(* Schneider Machine Expert - Basic project Schneider, file version 2.5.0.0 *)
(* ProjectInformations: Name=New project *)

HARDWARE
  Cpu 0: TM221CE24T
  EthernetConfiguration: NetworkName=M221, IpAllocationMode=FixedAddress, IpAddress=192.168.137.100, SubnetMask=255.255.255.0
  SerialLineConfiguration: Baud=Baud19200, Parity=ParityEven, DataBits=DataBits8, StopBits=StopBits1, PhysicalMedium=PhysicalMediumRs485, TransmissionMode=TransmissionModeModbusRtu, SlaveId=1, Addressing=SlaveAddressing
  MastTask: UsePeriodScanMode=false, PeriodScan=100
  FastTask: Period=255
  CpuBehavior: StartingMode=StartAsPreviousState, AutoSaveRamOnEeprom=true, WatchdogPeriod=250

SYMBOLS  (address, symbol, comment, settings)
  %MW1000   BLOCK1_START_TIME_Y  "BLOCK1 Start Time Years - 21"
  %MW1001   BLOCK1_START_TIME_M  "BLOCK1 Start Time  Months- 07"
  %MW1002   BLOCK1_START_TIME_D  "BLOCK1 Start Time Days- 19"
  %MW1003   BLOCK1_START_TIME_H  "BLOCK1 Start Time Hours - 14"
  %MW1004   BLOCK1_START_TIME_MN  "BLOCK1 Start Time Minutes - 33"
  %MW1007   BLOCK1_END_TIME_Y  "BLOCK1 End Time Years - 21"
  %MW1008   BLOCK1_END_TIME_M  "BLOCK1 End Time  Months- 07"
  %MW1009   BLOCK1_END_TIME_D  "BLOCK1 End Time Days- 19"
  %MW1010   BLOCK1_END_TIME_H  "BLOCK1 End Time Hours - 14"
  %MW1011   BLOCK1_END_TIME_MN  "BLOCK1 End Time Minutes - 33"
  %MW1012   BLOCK1_EC_SP_REAL  "BLOCK1 EC Setpoint"
  %MW1014   BLOCK1_RUNTIME_MN  "BLOCK1 Running Time for Cycle in Minutes"
  %MW1016   BLOCK1_TANK1_FLW_SP_REAL  "BLOCK1 Tank 1 Fertilizer Flow Setpoint"
  %MW1018   BLOCK1_TANK2_FLW_SP_REAL  "BLOCK1 Tank 2 Fertilizer Flow Setpoint"
  %MW1020   BLOCK1_TANK3_FLW_SP_REAL  "BLOCK1 Tank 3 Fertilizer Flow Setpoint"
  %MW1022   BLOCK1_TANK4_FLW_SP_REAL  "BLOCK1 Tank 4 Fertilizer Flow Setpoint"
  %MW1024   BLOCK1_TANK5_FLW_SP_REAL  "BLOCK1 Tank 5 Fertilizer Flow Setpoint"
  %MW1026   BLOCK1_TANK6_FLW_SP_REAL  "BLOCK1 Tank 6 Fertilizer Flow Setpoint"
  %MW1028   BLOCK1_TANK7_FLW_SP_REAL  "BLOCK1 Tank 7 Fertilizer Flow Setpoint"
  %MW1030   BLOCK1_TANK8_FLW_SP_REAL  "BLOCK1 Tank 8 Fertilizer Flow Setpoint"
  %MW1032   BLOCK1_TANK9_FLW_SP_REAL  "BLOCK1 Tank 9 Fertilizer Flow Setpoint"
  %MW1034   BLOCK1_TANK10_FLW_SP_REAL  "BLOCK1 Tank 10 Fertilizer Flow Setpoint"
  %MW1051   BLOCK2_START_TIME_Y  "BLOCK2 Start Time Years - 21"
  %MW1052   BLOCK2_START_TIME_M  "BLOCK2 Start Time  Months- 07"
  %MW1053   BLOCK2_START_TIME_D  "BLOCK2 Start Time Days- 19"
  %MW1054   BLOCK2_START_TIME_H  "BLOCK2 Start Time Hours - 14"
  %MW1055   BLOCK2_START_TIME_MN  "BLOCK2 Start Time Minutes - 33"
  %MW1058   BLOCK2_END_TIME_Y  "BLOCK2 End Time Years - 21"
  %MW1059   BLOCK2_END_TIME_M  "BLOCK2 End Time  Months- 07"
  %MW1060   BLOCK2_END_TIME_D  "BLOCK2 End Time Days- 19"
  %MW1061   BLOCK2_END_TIME_H  "BLOCK2 End Time Hours - 14"
  %MW1062   BLOCK2_END_TIME_MN  "BLOCK2 End Time Minutes - 33"
  %MW1063   BLOCK2_EC_SP_REAL  "BLOCK2 EC Setpoint"
  %MW1065   BLOCK2_RUNTIME_MN  "BLOCK2 Running Time for Cycle in Minutes"
  %MW1067   BLOCK2_TANK1_FLW_SP_REAL  "BLOCK2 Tank 1 Fertilizer Flow Setpoint"
  %MW1069   BLOCK2_TANK2_FLW_SP_REAL  "BLOCK2 Tank 2 Fertilizer Flow Setpoint"
  %MW1071   BLOCK2_TANK3_FLW_SP_REAL  "BLOCK2 Tank 3 Fertilizer Flow Setpoint"
  %MW1073   BLOCK2_TANK4_FLW_SP_REAL  "BLOCK2 Tank 4 Fertilizer Flow Setpoint"
  %MW1075   BLOCK2_TANK5_FLW_SP_REAL  "BLOCK2 Tank 5 Fertilizer Flow Setpoint"
  %MW1077   BLOCK2_TANK6_FLW_SP_REAL  "BLOCK2 Tank 6 Fertilizer Flow Setpoint"
  %MW1079   BLOCK2_TANK7_FLW_SP_REAL  "BLOCK2 Tank 7 Fertilizer Flow Setpoint"
  %MW1081   BLOCK2_TANK8_FLW_SP_REAL  "BLOCK2 Tank 8 Fertilizer Flow Setpoint"
  %MW1083   BLOCK2_TANK9_FLW_SP_REAL  "BLOCK2 Tank 9 Fertilizer Flow Setpoint"
  %MW1085   BLOCK2_TANK10_FLW_SP_REAL  "BLOCK2 Tank 10 Fertilizer Flow Setpoint"
  %MW1102   BLOCK3_START_TIME_Y  "BLOCK3 Start Time Years - 21"
  %MW1103   BLOCK3_START_TIME_M  "BLOCK3 Start Time  Months- 07"
  %MW1104   BLOCK3_START_TIME_D  "BLOCK3 Start Time Days- 19"
  %MW1105   BLOCK3_START_TIME_H  "BLOCK3 Start Time Hours - 14"
  %MW1106   BLOCK3_START_TIME_MN  "BLOCK3 Start Time Minutes - 33"
  %MW1109   BLOCK3_END_TIME_Y  "BLOCK3 End Time Years - 21"
  %MW1110   BLOCK3_END_TIME_M  "BLOCK3 End Time  Months- 07"
  %MW1111   BLOCK3_END_TIME_D  "BLOCK3 End Time Days- 19"
  %MW1112   BLOCK3_END_TIME_H  "BLOCK3 End Time Hours - 14"
  %MW1113   BLOCK3_END_TIME_MN  "BLOCK3 End Time Minutes - 33"
  %MW1114   BLOCK3_EC_SP_REAL  "BLOCK3 EC Setpoint"
  %MW1116   BLOCK3_RUNTIME_MN  "BLOCK3 Running Time for Cycle in Minutes"
  %MW1118   BLOCK3_TANK1_FLW_SP_REAL  "BLOCK3 Tank 1 Fertilizer Flow Setpoint"
  %MW1120   BLOCK3_TANK2_FLW_SP_REAL  "BLOCK3 Tank 2 Fertilizer Flow Setpoint"
  %MW1122   BLOCK3_TANK3_FLW_SP_REAL  "BLOCK3 Tank 3 Fertilizer Flow Setpoint"
  %MW1124   BLOCK3_TANK4_FLW_SP_REAL  "BLOCK3 Tank 4 Fertilizer Flow Setpoint"
  %MW1126   BLOCK3_TANK5_FLW_SP_REAL  "BLOCK3 Tank 5 Fertilizer Flow Setpoint"
  %MW1128   BLOCK3_TANK6_FLW_SP_REAL  "BLOCK3 Tank 6 Fertilizer Flow Setpoint"
  %MW1130   BLOCK3_TANK7_FLW_SP_REAL  "BLOCK3 Tank 7 Fertilizer Flow Setpoint"
  %MW1132   BLOCK3_TANK8_FLW_SP_REAL  "BLOCK3 Tank 8 Fertilizer Flow Setpoint"
  %MW1134   BLOCK3_TANK9_FLW_SP_REAL  "BLOCK3 Tank 9 Fertilizer Flow Setpoint"
  %MW1136   BLOCK3_TANK10_FLW_SP_REAL  "BLOCK3 Tank 10 Fertilizer Flow Setpoint"
  %MW1153   BLOCK4_START_TIME_Y  "BLOCK4 Start Time Years - 21"
  %MW1154   BLOCK4_START_TIME_M  "BLOCK4 Start Time  Months- 07"
  %MW1155   BLOCK4_START_TIME_D  "BLOCK4 Start Time Days- 19"
  %MW1156   BLOCK4_START_TIME_H  "BLOCK4 Start Time Hours - 14"
  %MW1157   BLOCK4_START_TIME_MN  "BLOCK4 Start Time Minutes - 33"
  %MW1160   BLOCK4_END_TIME_Y  "BLOCK4 End Time Years - 21"
  %MW1161   BLOCK4_END_TIME_M  "BLOCK4 End Time  Months- 07"
  %MW1162   BLOCK4_END_TIME_D  "BLOCK4 End Time Days- 19"
  %MW1163   BLOCK4_END_TIME_H  "BLOCK4 End Time Hours - 14"
  %MW1164   BLOCK4_END_TIME_MN  "BLOCK4 End Time Minutes - 33"
  %MW1165   BLOCK4_EC_SP_REAL  "BLOCK4 EC Setpoint"
  %MW1167   BLOCK4_RUNTIME_MN  "BLOCK4 Running Time for Cycle in Minutes"
  %MW1169   BLOCK4_TANK1_FLW_SP_REAL  "BLOCK4 Tank 1 Fertilizer Flow Setpoint"
  %MW1171   BLOCK4_TANK2_FLW_SP_REAL  "BLOCK4 Tank 2 Fertilizer Flow Setpoint"
  %MW1173   BLOCK4_TANK3_FLW_SP_REAL  "BLOCK4 Tank 3 Fertilizer Flow Setpoint"
  %MW1175   BLOCK4_TANK4_FLW_SP_REAL  "BLOCK4 Tank 4 Fertilizer Flow Setpoint"
  %MW1177   BLOCK4_TANK5_FLW_SP_REAL  "BLOCK4 Tank 5 Fertilizer Flow Setpoint"
  %MW1179   BLOCK4_TANK6_FLW_SP_REAL  "BLOCK4 Tank 6 Fertilizer Flow Setpoint"
  %MW1181   BLOCK4_TANK7_FLW_SP_REAL  "BLOCK4 Tank 7 Fertilizer Flow Setpoint"
  %MW1183   BLOCK4_TANK8_FLW_SP_REAL  "BLOCK4 Tank 8 Fertilizer Flow Setpoint"
  %MW1185   BLOCK4_TANK9_FLW_SP_REAL  "BLOCK4 Tank 9 Fertilizer Flow Setpoint"
  %MW1187   BLOCK4_TANK10_FLW_SP_REAL  "BLOCK4 Tank 10 Fertilizer Flow Setpoint"
  %MW1204   BLOCK5_START_TIME_Y  "BLOCK5 Start Time Years - 21"
  %MW1205   BLOCK5_START_TIME_M  "BLOCK5 Start Time  Months- 07"
  %MW1206   BLOCK5_START_TIME_D  "BLOCK5 Start Time Days- 19"
  %MW1207   BLOCK5_START_TIME_H  "BLOCK5 Start Time Hours - 14"
  %MW1208   BLOCK5_START_TIME_MN  "BLOCK5 Start Time Minutes - 33"
  %MW1211   BLOCK5_END_TIME_Y  "BLOCK5 End Time Years - 21"
  %MW1212   BLOCK5_END_TIME_M  "BLOCK5 End Time  Months- 07"
  %MW1213   BLOCK5_END_TIME_D  "BLOCK5 End Time Days- 19"
  %MW1214   BLOCK5_END_TIME_H  "BLOCK5 End Time Hours - 14"
  %MW1215   BLOCK5_END_TIME_MN  "BLOCK5 End Time Minutes - 33"
  %MW1216   BLOCK5_EC_SP_REAL  "BLOCK5 EC Setpoint"
  %MW1218   BLOCK5_RUNTIME_MN  "BLOCK5 Running Time for Cycle in Minutes"
  %MW1220   BLOCK5_TANK1_FLW_SP_REAL  "BLOCK5 Tank 1 Fertilizer Flow Setpoint"
  %MW1222   BLOCK5_TANK2_FLW_SP_REAL  "BLOCK5 Tank 2 Fertilizer Flow Setpoint"
  %MW1224   BLOCK5_TANK3_FLW_SP_REAL  "BLOCK5 Tank 3 Fertilizer Flow Setpoint"
  %MW1226   BLOCK5_TANK4_FLW_SP_REAL  "BLOCK5 Tank 4 Fertilizer Flow Setpoint"
  %MW1228   BLOCK5_TANK5_FLW_SP_REAL  "BLOCK5 Tank 5 Fertilizer Flow Setpoint"
  %MW1230   BLOCK5_TANK6_FLW_SP_REAL  "BLOCK5 Tank 6 Fertilizer Flow Setpoint"
  %MW1232   BLOCK5_TANK7_FLW_SP_REAL  "BLOCK5 Tank 7 Fertilizer Flow Setpoint"
  %MW1234   BLOCK5_TANK8_FLW_SP_REAL  "BLOCK5 Tank 8 Fertilizer Flow Setpoint"
  %MW1236   BLOCK5_TANK9_FLW_SP_REAL  "BLOCK5 Tank 9 Fertilizer Flow Setpoint"
  %MW1238   BLOCK5_TANK10_FLW_SP_REAL  "BLOCK5 Tank 10 Fertilizer Flow Setpoint"
  %MW1255   BLOCK6_START_TIME_Y  "BLOCK6 Start Time Years - 21"
  %MW1256   BLOCK6_START_TIME_M  "BLOCK6 Start Time  Months- 07"
  %MW1257   BLOCK6_START_TIME_D  "BLOCK6 Start Time Days- 19"
  %MW1258   BLOCK6_START_TIME_H  "BLOCK6 Start Time Hours - 14"
  %MW1259   BLOCK6_START_TIME_MN  "BLOCK6 Start Time Minutes - 33"
  %MW1262   BLOCK6_END_TIME_Y  "BLOCK6 End Time Years - 21"
  %MW1263   BLOCK6_END_TIME_M  "BLOCK6 End Time  Months- 07"
  %MW1264   BLOCK6_END_TIME_D  "BLOCK6 End Time Days- 19"
  %MW1265   BLOCK6_END_TIME_H  "BLOCK6 End Time Hours - 14"
  %MW1266   BLOCK6_END_TIME_MN  "BLOCK6 End Time Minutes - 33"
  %MW1267   BLOCK6_EC_SP_REAL  "BLOCK6 EC Setpoint"
  %MW1269   BLOCK6_RUNTIME_MN  "BLOCK6 Running Time for Cycle in Minutes"
  %MW1271   BLOCK6_TANK1_FLW_SP_REAL  "BLOCK6 Tank 1 Fertilizer Flow Setpoint"
  %MW1273   BLOCK6_TANK2_FLW_SP_REAL  "BLOCK6 Tank 2 Fertilizer Flow Setpoint"
  %MW1275   BLOCK6_TANK3_FLW_SP_REAL  "BLOCK6 Tank 3 Fertilizer Flow Setpoint"
  %MW1277   BLOCK6_TANK4_FLW_SP_REAL  "BLOCK6 Tank 4 Fertilizer Flow Setpoint"
  %MW1279   BLOCK6_TANK5_FLW_SP_REAL  "BLOCK6 Tank 5 Fertilizer Flow Setpoint"
  %MW1281   BLOCK6_TANK6_FLW_SP_REAL  "BLOCK6 Tank 6 Fertilizer Flow Setpoint"
  %MW1283   BLOCK6_TANK7_FLW_SP_REAL  "BLOCK6 Tank 7 Fertilizer Flow Setpoint"
  %MW1285   BLOCK6_TANK8_FLW_SP_REAL  "BLOCK6 Tank 8 Fertilizer Flow Setpoint"
  %MW1287   BLOCK6_TANK9_FLW_SP_REAL  "BLOCK6 Tank 9 Fertilizer Flow Setpoint"
  %MW1289   BLOCK6_TANK10_FLW_SP_REAL  "BLOCK6 Tank 10 Fertilizer Flow Setpoint"
  %MW1306   BLOCK7_START_TIME_Y  "BLOCK7 Start Time Years - 21"
  %MW1307   BLOCK7_START_TIME_M  "BLOCK7 Start Time  Months- 07"
  %MW1308   BLOCK7_START_TIME_D  "BLOCK7 Start Time Days- 19"
  %MW1309   BLOCK7_START_TIME_H  "BLOCK7 Start Time Hours - 14"
  %MW1310   BLOCK7_START_TIME_MN  "BLOCK7 Start Time Minutes - 33"
  %MW1313   BLOCK7_END_TIME_Y  "BLOCK7 End Time Years - 21"
  %MW1314   BLOCK7_END_TIME_M  "BLOCK7 End Time  Months- 07"
  %MW1315   BLOCK7_END_TIME_D  "BLOCK7 End Time Days- 19"
  %MW1316   BLOCK7_END_TIME_H  "BLOCK7 End Time Hours - 14"
  %MW1317   BLOCK7_END_TIME_MN  "BLOCK7 End Time Minutes - 33"
  %MW1318   BLOCK7_EC_SP_REAL  "BLOCK7 EC Setpoint"
  %MW1320   BLOCK7_RUNTIME_MN  "BLOCK7 Running Time for Cycle in Minutes"
  %MW1322   BLOCK7_TANK1_FLW_SP_REAL  "BLOCK7 Tank 1 Fertilizer Flow Setpoint"
  %MW1324   BLOCK7_TANK2_FLW_SP_REAL  "BLOCK7 Tank 2 Fertilizer Flow Setpoint"
  %MW1326   BLOCK7_TANK3_FLW_SP_REAL  "BLOCK7 Tank 3 Fertilizer Flow Setpoint"
  %MW1328   BLOCK7_TANK4_FLW_SP_REAL  "BLOCK7 Tank 4 Fertilizer Flow Setpoint"
  %MW1330   BLOCK7_TANK5_FLW_SP_REAL  "BLOCK7 Tank 5 Fertilizer Flow Setpoint"
  %MW1332   BLOCK7_TANK6_FLW_SP_REAL  "BLOCK7 Tank 6 Fertilizer Flow Setpoint"
  %MW1334   BLOCK7_TANK7_FLW_SP_REAL  "BLOCK7 Tank 7 Fertilizer Flow Setpoint"
  %MW1336   BLOCK7_TANK8_FLW_SP_REAL  "BLOCK7 Tank 8 Fertilizer Flow Setpoint"
  %MW1338   BLOCK7_TANK9_FLW_SP_REAL  "BLOCK7 Tank 9 Fertilizer Flow Setpoint"
  %MW1340   BLOCK7_TANK10_FLW_SP_REAL  "BLOCK7 Tank 10 Fertilizer Flow Setpoint"
  %MW1357   BLOCK8_START_TIME_Y  "BLOCK8 Start Time Years - 21"
  %MW1358   BLOCK8_START_TIME_M  "BLOCK8 Start Time  Months- 07"
  %MW1359   BLOCK8_START_TIME_D  "BLOCK8 Start Time Days- 19"
  %MW1360   BLOCK8_START_TIME_H  "BLOCK8 Start Time Hours - 14"
  %MW1361   BLOCK8_START_TIME_MN  "BLOCK8 Start Time Minutes - 33"
  %MW1364   BLOCK8_END_TIME_Y  "BLOCK8 End Time Years - 21"
  %MW1365   BLOCK8_END_TIME_M  "BLOCK8 End Time  Months- 07"
  %MW1366   BLOCK8_END_TIME_D  "BLOCK8 End Time Days- 19"
  %MW1367   BLOCK8_END_TIME_H  "BLOCK8 End Time Hours - 14"
  %MW1368   BLOCK8_END_TIME_MN  "BLOCK8 End Time Minutes - 33"
  %MW1369   BLOCK8_EC_SP_REAL  "BLOCK8 EC Setpoint"
  %MW1371   BLOCK8_RUNTIME_MN  "BLOCK8 Running Time for Cycle in Minutes"
  %MW1373   BLOCK8_TANK1_FLW_SP_REAL  "BLOCK8 Tank 1 Fertilizer Flow Setpoint"
  %MW1375   BLOCK8_TANK2_FLW_SP_REAL  "BLOCK8 Tank 2 Fertilizer Flow Setpoint"
  %MW1377   BLOCK8_TANK3_FLW_SP_REAL  "BLOCK8 Tank 3 Fertilizer Flow Setpoint"
  %MW1379   BLOCK8_TANK4_FLW_SP_REAL  "BLOCK8 Tank 4 Fertilizer Flow Setpoint"
  %MW1381   BLOCK8_TANK5_FLW_SP_REAL  "BLOCK8 Tank 5 Fertilizer Flow Setpoint"
  %MW1383   BLOCK8_TANK6_FLW_SP_REAL  "BLOCK8 Tank 6 Fertilizer Flow Setpoint"
  %MW1385   BLOCK8_TANK7_FLW_SP_REAL  "BLOCK8 Tank 7 Fertilizer Flow Setpoint"
  %MW1387   BLOCK8_TANK8_FLW_SP_REAL  "BLOCK8 Tank 8 Fertilizer Flow Setpoint"
  %MW1389   BLOCK8_TANK9_FLW_SP_REAL  "BLOCK8 Tank 9 Fertilizer Flow Setpoint"
  %MW1391   BLOCK8_TANK10_FLW_SP_REAL  "BLOCK8 Tank 10 Fertilizer Flow Setpoint"
  %MW1408   BLOCK9_START_TIME_Y  "BLOCK9 Start Time Years - 21"
  %MW1409   BLOCK9_START_TIME_M  "BLOCK9 Start Time  Months- 07"
  %MW1410   BLOCK9_START_TIME_D  "BLOCK9 Start Time Days- 19"
  %MW1411   BLOCK9_START_TIME_H  "BLOCK9 Start Time Hours - 14"
  %MW1412   BLOCK9_START_TIME_MN  "BLOCK9 Start Time Minutes - 33"
  %MW1415   BLOCK9_END_TIME_Y  "BLOCK9 End Time Years - 21"
  %MW1416   BLOCK9_END_TIME_M  "BLOCK9 End Time  Months- 07"
  %MW1417   BLOCK9_END_TIME_D  "BLOCK9 End Time Days- 19"
  %MW1418   BLOCK9_END_TIME_H  "BLOCK9 End Time Hours - 14"
  %MW1419   BLOCK9_END_TIME_MN  "BLOCK9 End Time Minutes - 33"
  %MW1420   BLOCK9_EC_SP_REAL  "BLOCK9 EC Setpoint"
  %MW1422   BLOCK9_RUNTIME_MN  "BLOCK9 Running Time for Cycle in Minutes"
  %MW1424   BLOCK9_TANK1_FLW_SP_REAL  "BLOCK9 Tank 1 Fertilizer Flow Setpoint"
  %MW1426   BLOCK9_TANK2_FLW_SP_REAL  "BLOCK9 Tank 2 Fertilizer Flow Setpoint"
  %MW1428   BLOCK9_TANK3_FLW_SP_REAL  "BLOCK9 Tank 3 Fertilizer Flow Setpoint"
  %MW1430   BLOCK9_TANK4_FLW_SP_REAL  "BLOCK9 Tank 4 Fertilizer Flow Setpoint"
  %MW1432   BLOCK9_TANK5_FLW_SP_REAL  "BLOCK9 Tank 5 Fertilizer Flow Setpoint"
  %MW1434   BLOCK9_TANK6_FLW_SP_REAL  "BLOCK9 Tank 6 Fertilizer Flow Setpoint"
  %MW1436   BLOCK9_TANK7_FLW_SP_REAL  "BLOCK9 Tank 7 Fertilizer Flow Setpoint"
  %MW1438   BLOCK9_TANK8_FLW_SP_REAL  "BLOCK9 Tank 8 Fertilizer Flow Setpoint"
  %MW1440   BLOCK9_TANK9_FLW_SP_REAL  "BLOCK9 Tank 9 Fertilizer Flow Setpoint"
  %MW1442   BLOCK9_TANK10_FLW_SP_REAL  "BLOCK9 Tank 10 Fertilizer Flow Setpoint"
  %MW1459   BLOCK10_START_TIME_Y  "BLOCK10 Start Time Years - 21"
  %MW1460   BLOCK10_START_TIME_M  "BLOCK10 Start Time  Months- 07"
  %MW1461   BLOCK10_START_TIME_D  "BLOCK10 Start Time Days- 19"
  %MW1462   BLOCK10_START_TIME_H  "BLOCK10 Start Time Hours - 14"
  %MW1463   BLOCK10_START_TIME_MN  "BLOCK10 Start Time Minutes - 33"
  %MW1466   BLOCK10_END_TIME_Y  "BLOCK10 End Time Years - 21"
  %MW1467   BLOCK10_END_TIME_M  "BLOCK10 End Time  Months- 07"
  %MW1468   BLOCK10_END_TIME_D  "BLOCK10 End Time Days- 19"
  %MW1469   BLOCK10_END_TIME_H  "BLOCK10 End Time Hours - 14"
  %MW1470   BLOCK10_END_TIME_MN  "BLOCK10 End Time Minutes - 33"
  %MW1471   BLOCK10_EC_SP_REAL  "BLOCK10 EC Setpoint"
  %MW1473   BLOCK10_RUNTIME_MN  "BLOCK10 Running Time for Cycle in Minutes"
  %MW1475   BLOCK10_TANK1_FLW_SP_REAL  "BLOCK10 Tank 1 Fertilizer Flow Setpoint"
  %MW1477   BLOCK10_TANK2_FLW_SP_REAL  "BLOCK10 Tank 2 Fertilizer Flow Setpoint"
  %MW1479   BLOCK10_TANK3_FLW_SP_REAL  "BLOCK10 Tank 3 Fertilizer Flow Setpoint"
  %MW1481   BLOCK10_TANK4_FLW_SP_REAL  "BLOCK10 Tank 4 Fertilizer Flow Setpoint"
  %MW1483   BLOCK10_TANK5_FLW_SP_REAL  "BLOCK10 Tank 5 Fertilizer Flow Setpoint"
  %MW1485   BLOCK10_TANK6_FLW_SP_REAL  "BLOCK10 Tank 6 Fertilizer Flow Setpoint"
  %MW1487   BLOCK10_TANK7_FLW_SP_REAL  "BLOCK10 Tank 7 Fertilizer Flow Setpoint"
  %MW1489   BLOCK10_TANK8_FLW_SP_REAL  "BLOCK10 Tank 8 Fertilizer Flow Setpoint"
  %MW1491   BLOCK10_TANK9_FLW_SP_REAL  "BLOCK10 Tank 9 Fertilizer Flow Setpoint"
  %MW1493   BLOCK10_TANK10_FLW_SP_REAL  "BLOCK10 Tank 10 Fertilizer Flow Setpoint"
  %MW1510   BLOCK11_START_TIME_Y  "BLOCK11 Start Time Years - 21"
  %MW1511   BLOCK11_START_TIME_M  "BLOCK11 Start Time  Months- 07"
  %MW1512   BLOCK11_START_TIME_D  "BLOCK11 Start Time Days- 19"
  %MW1513   BLOCK11_START_TIME_H  "BLOCK11 Start Time Hours - 14"
  %MW1514   BLOCK11_START_TIME_MN  "BLOCK11 Start Time Minutes - 33"
  %MW1517   BLOCK11_END_TIME_Y  "BLOCK11 End Time Years - 21"
  %MW1518   BLOCK11_END_TIME_M  "BLOCK11 End Time  Months- 07"
  %MW1519   BLOCK11_END_TIME_D  "BLOCK11 End Time Days- 19"
  %MW1520   BLOCK11_END_TIME_H  "BLOCK11 End Time Hours - 14"
  %MW1521   BLOCK11_END_TIME_MN  "BLOCK11 End Time Minutes - 33"
  %MW1522   BLOCK11_EC_SP_REAL  "BLOCK11 EC Setpoint"
  %MW1524   BLOCK11_RUNTIME_MN  "BLOCK11 Running Time for Cycle in Minutes"
  %MW1526   BLOCK11_TANK1_FLW_SP_REAL  "BLOCK11 Tank 1 Fertilizer Flow Setpoint"
  %MW1528   BLOCK11_TANK2_FLW_SP_REAL  "BLOCK11 Tank 2 Fertilizer Flow Setpoint"
  %MW1530   BLOCK11_TANK3_FLW_SP_REAL  "BLOCK11 Tank 3 Fertilizer Flow Setpoint"
  %MW1532   BLOCK11_TANK4_FLW_SP_REAL  "BLOCK11 Tank 4 Fertilizer Flow Setpoint"
  %MW1534   BLOCK11_TANK5_FLW_SP_REAL  "BLOCK11 Tank 5 Fertilizer Flow Setpoint"
  %MW1536   BLOCK11_TANK6_FLW_SP_REAL  "BLOCK11 Tank 6 Fertilizer Flow Setpoint"
  %MW1538   BLOCK11_TANK7_FLW_SP_REAL  "BLOCK11 Tank 7 Fertilizer Flow Setpoint"
  %MW1540   BLOCK11_TANK8_FLW_SP_REAL  "BLOCK11 Tank 8 Fertilizer Flow Setpoint"
  %MW1542   BLOCK11_TANK9_FLW_SP_REAL  "BLOCK11 Tank 9 Fertilizer Flow Setpoint"
  %MW1544   BLOCK11_TANK10_FLW_SP_REAL  "BLOCK11 Tank 10 Fertilizer Flow Setpoint"
  %MW1561   BLOCK12_START_TIME_Y  "BLOCK12 Start Time Years - 21"
  %MW1562   BLOCK12_START_TIME_M  "BLOCK12 Start Time  Months- 07"
  %MW1563   BLOCK12_START_TIME_D  "BLOCK12 Start Time Days- 19"
  %MW1564   BLOCK12_START_TIME_H  "BLOCK12 Start Time Hours - 14"
  %MW1565   BLOCK12_START_TIME_MN  "BLOCK12 Start Time Minutes - 33"
  %MW1568   BLOCK12_END_TIME_Y  "BLOCK12 End Time Years - 21"
  %MW1569   BLOCK12_END_TIME_M  "BLOCK12 End Time  Months- 07"
  %MW1570   BLOCK12_END_TIME_D  "BLOCK12 End Time Days- 19"
  %MW1571   BLOCK12_END_TIME_H  "BLOCK12 End Time Hours - 14"
  %MW1572   BLOCK12_END_TIME_MN  "BLOCK12 End Time Minutes - 33"
  %MW1573   BLOCK12_EC_SP_REAL  "BLOCK12 EC Setpoint"
  %MW1575   BLOCK12_RUNTIME_MN  "BLOCK12 Running Time for Cycle in Minutes"
  %MW1577   BLOCK12_TANK1_FLW_SP_REAL  "BLOCK12 Tank 1 Fertilizer Flow Setpoint"
  %MW1579   BLOCK12_TANK2_FLW_SP_REAL  "BLOCK12 Tank 2 Fertilizer Flow Setpoint"
  %MW1581   BLOCK12_TANK3_FLW_SP_REAL  "BLOCK12 Tank 3 Fertilizer Flow Setpoint"
  %MW1583   BLOCK12_TANK4_FLW_SP_REAL  "BLOCK12 Tank 4 Fertilizer Flow Setpoint"
  %MW1585   BLOCK12_TANK5_FLW_SP_REAL  "BLOCK12 Tank 5 Fertilizer Flow Setpoint"
  %MW1587   BLOCK12_TANK6_FLW_SP_REAL  "BLOCK12 Tank 6 Fertilizer Flow Setpoint"
  %MW1589   BLOCK12_TANK7_FLW_SP_REAL  "BLOCK12 Tank 7 Fertilizer Flow Setpoint"
  %MW1591   BLOCK12_TANK8_FLW_SP_REAL  "BLOCK12 Tank 8 Fertilizer Flow Setpoint"
  %MW1593   BLOCK12_TANK9_FLW_SP_REAL  "BLOCK12 Tank 9 Fertilizer Flow Setpoint"
  %MW1595   BLOCK12_TANK10_FLW_SP_REAL  "BLOCK12 Tank 10 Fertilizer Flow Setpoint"
  %MW1612   BLOCK13_START_TIME_Y  "BLOCK13 Start Time Years - 21"
  %MW1613   BLOCK13_START_TIME_M  "BLOCK13 Start Time  Months- 07"
  %MW1614   BLOCK13_START_TIME_D  "BLOCK13 Start Time Days- 19"
  %MW1615   BLOCK13_START_TIME_H  "BLOCK13 Start Time Hours - 14"
  %MW1616   BLOCK13_START_TIME_MN  "BLOCK13 Start Time Minutes - 33"
  %MW1619   BLOCK13_END_TIME_Y  "BLOCK13 End Time Years - 21"
  %MW1620   BLOCK13_END_TIME_M  "BLOCK13 End Time  Months- 07"
  %MW1621   BLOCK13_END_TIME_D  "BLOCK13 End Time Days- 19"
  %MW1622   BLOCK13_END_TIME_H  "BLOCK13 End Time Hours - 14"
  %MW1623   BLOCK13_END_TIME_MN  "BLOCK13 End Time Minutes - 33"
  %MW1624   BLOCK13_EC_SP_REAL  "BLOCK13 EC Setpoint"
  %MW1626   BLOCK13_RUNTIME_MN  "BLOCK13 Running Time for Cycle in Minutes"
  %MW1628   BLOCK13_TANK1_FLW_SP_REAL  "BLOCK13 Tank 1 Fertilizer Flow Setpoint"
  %MW1630   BLOCK13_TANK2_FLW_SP_REAL  "BLOCK13 Tank 2 Fertilizer Flow Setpoint"
  %MW1632   BLOCK13_TANK3_FLW_SP_REAL  "BLOCK13 Tank 3 Fertilizer Flow Setpoint"
  %MW1634   BLOCK13_TANK4_FLW_SP_REAL  "BLOCK13 Tank 4 Fertilizer Flow Setpoint"
  %MW1636   BLOCK13_TANK5_FLW_SP_REAL  "BLOCK13 Tank 5 Fertilizer Flow Setpoint"
  %MW1638   BLOCK13_TANK6_FLW_SP_REAL  "BLOCK13 Tank 6 Fertilizer Flow Setpoint"
  %MW1640   BLOCK13_TANK7_FLW_SP_REAL  "BLOCK13 Tank 7 Fertilizer Flow Setpoint"
  %MW1642   BLOCK13_TANK8_FLW_SP_REAL  "BLOCK13 Tank 8 Fertilizer Flow Setpoint"
  %MW1644   BLOCK13_TANK9_FLW_SP_REAL  "BLOCK13 Tank 9 Fertilizer Flow Setpoint"
  %MW1646   BLOCK13_TANK10_FLW_SP_REAL  "BLOCK13 Tank 10 Fertilizer Flow Setpoint"
  %MW1663   BLOCK14_START_TIME_Y  "BLOCK14 Start Time Years - 21"
  %MW1664   BLOCK14_START_TIME_M  "BLOCK14 Start Time  Months- 07"
  %MW1665   BLOCK14_START_TIME_D  "BLOCK14 Start Time Days- 19"
  %MW1666   BLOCK14_START_TIME_H  "BLOCK14 Start Time Hours - 14"
  %MW1667   BLOCK14_START_TIME_MN  "BLOCK14 Start Time Minutes - 33"
  %MW1670   BLOCK14_END_TIME_Y  "BLOCK14 End Time Years - 21"
  %MW1671   BLOCK14_END_TIME_M  "BLOCK14 End Time  Months- 07"
  %MW1672   BLOCK14_END_TIME_D  "BLOCK14 End Time Days- 19"
  %MW1673   BLOCK14_END_TIME_H  "BLOCK14 End Time Hours - 14"
  %MW1674   BLOCK14_END_TIME_MN  "BLOCK14 End Time Minutes - 33"
  %MW1675   BLOCK14_EC_SP_REAL  "BLOCK14 EC Setpoint"
  %MW1677   BLOCK14_RUNTIME_MN  "BLOCK14 Running Time for Cycle in Minutes"
  %MW1679   BLOCK14_TANK1_FLW_SP_REAL  "BLOCK14 Tank 1 Fertilizer Flow Setpoint"
  %MW1681   BLOCK14_TANK2_FLW_SP_REAL  "BLOCK14 Tank 2 Fertilizer Flow Setpoint"
  %MW1683   BLOCK14_TANK3_FLW_SP_REAL  "BLOCK14 Tank 3 Fertilizer Flow Setpoint"
  %MW1685   BLOCK14_TANK4_FLW_SP_REAL  "BLOCK14 Tank 4 Fertilizer Flow Setpoint"
  %MW1687   BLOCK14_TANK5_FLW_SP_REAL  "BLOCK14 Tank 5 Fertilizer Flow Setpoint"
  %MW1689   BLOCK14_TANK6_FLW_SP_REAL  "BLOCK14 Tank 6 Fertilizer Flow Setpoint"
  %MW1691   BLOCK14_TANK7_FLW_SP_REAL  "BLOCK14 Tank 7 Fertilizer Flow Setpoint"
  %MW1693   BLOCK14_TANK8_FLW_SP_REAL  "BLOCK14 Tank 8 Fertilizer Flow Setpoint"
  %MW1695   BLOCK14_TANK9_FLW_SP_REAL  "BLOCK14 Tank 9 Fertilizer Flow Setpoint"
  %MW1697   BLOCK14_TANK10_FLW_SP_REAL  "BLOCK14 Tank 10 Fertilizer Flow Setpoint"
  %MW1714   BLOCK15_START_TIME_Y  "BLOCK15 Start Time Years - 21"
  %MW1715   BLOCK15_START_TIME_M  "BLOCK15 Start Time  Months- 07"
  %MW1716   BLOCK15_START_TIME_D  "BLOCK15 Start Time Days- 19"
  %MW1717   BLOCK15_START_TIME_H  "BLOCK15 Start Time Hours - 14"
  %MW1718   BLOCK15_START_TIME_MN  "BLOCK15 Start Time Minutes - 33"
  %MW1721   BLOCK15_END_TIME_Y  "BLOCK15 End Time Years - 21"
  %MW1722   BLOCK15_END_TIME_M  "BLOCK15 End Time  Months- 07"
  %MW1723   BLOCK15_END_TIME_D  "BLOCK15 End Time Days- 19"
  %MW1724   BLOCK15_END_TIME_H  "BLOCK15 End Time Hours - 14"
  %MW1725   BLOCK15_END_TIME_MN  "BLOCK15 End Time Minutes - 33"
  %MW1726   BLOCK15_EC_SP_REAL  "BLOCK15 EC Setpoint"
  %MW1728   BLOCK15_RUNTIME_MN  "BLOCK15 Running Time for Cycle in Minutes"
  %MW1730   BLOCK15_TANK1_FLW_SP_REAL  "BLOCK15 Tank 1 Fertilizer Flow Setpoint"
  %MW1732   BLOCK15_TANK2_FLW_SP_REAL  "BLOCK15 Tank 2 Fertilizer Flow Setpoint"
  %MW1734   BLOCK15_TANK3_FLW_SP_REAL  "BLOCK15 Tank 3 Fertilizer Flow Setpoint"
  %MW1736   BLOCK15_TANK4_FLW_SP_REAL  "BLOCK15 Tank 4 Fertilizer Flow Setpoint"
  %MW1738   BLOCK15_TANK5_FLW_SP_REAL  "BLOCK15 Tank 5 Fertilizer Flow Setpoint"
  %MW1740   BLOCK15_TANK6_FLW_SP_REAL  "BLOCK15 Tank 6 Fertilizer Flow Setpoint"
  %MW1742   BLOCK15_TANK7_FLW_SP_REAL  "BLOCK15 Tank 7 Fertilizer Flow Setpoint"
  %MW1744   BLOCK15_TANK8_FLW_SP_REAL  "BLOCK15 Tank 8 Fertilizer Flow Setpoint"
  %MW1746   BLOCK15_TANK9_FLW_SP_REAL  "BLOCK15 Tank 9 Fertilizer Flow Setpoint"
  %MW1748   BLOCK15_TANK10_FLW_SP_REAL  "BLOCK15 Tank 10 Fertilizer Flow Setpoint"
  %MW1750   BLOCK27_START_TIME_Y  "BLOCK27 Start Time Years - 21"
  %MW1751   BLOCK27_START_TIME_M  "BLOCK27 Start Time  Months- 07"
  %MW1752   BLOCK27_START_TIME_D  "BLOCK27 Start Time Days- 19"
  %MW1753   BLOCK27_START_TIME_H  "BLOCK27 Start Time Hours - 14"
  %MW1754   BLOCK27_START_TIME_MN  "BLOCK27 Start Time Minutes - 33"
  %MW1755   BLOCK27_SPARE_01
  %MW1756   BLOCK27_SPARE_02
  %MW1757   BLOCK27_END_TIME_Y  "BLOCK27 End Time Years - 21"
  %MW1758   BLOCK27_END_TIME_M  "BLOCK27 End Time  Months- 07"
  %MW1759   BLOCK27_END_TIME_D  "BLOCK27 End Time Days- 19"
  %MW1760   BLOCK27_END_TIME_H  "BLOCK27 End Time Hours - 14"
  %MW1761   BLOCK27_END_TIME_MN  "BLOCK27 End Time Minutes - 33"
  %MW1762   BLOCK27_SPARE_03
  %MW1763   BLOCK27_SPARE_04
  %MW1764   BLOCK27_RUNTIME_MN  "BLOCK27 Running Time for Cycle in Minutes"
  %MW1780   BLOCK28_START_TIME_Y  "BLOCK28 Start Time Years - 21"
  %MW1781   BLOCK28_START_TIME_M  "BLOCK28 Start Time  Months- 07"
  %MW1782   BLOCK28_START_TIME_D  "BLOCK28 Start Time Days- 19"
  %MW1783   BLOCK28_START_TIME_H  "BLOCK28 Start Time Hours - 14"
  %MW1784   BLOCK28_START_TIME_MN  "BLOCK28 Start Time Minutes - 33"
  %MW1785   BLOCK28_SPARE_01
  %MW1786   BLOCK28_SPARE_02
  %MW1787   BLOCK28_END_TIME_Y  "BLOCK28 End Time Years - 21"
  %MW1788   BLOCK28_END_TIME_M  "BLOCK28 End Time  Months- 07"
  %MW1789   BLOCK28_END_TIME_D  "BLOCK28 End Time Days- 19"
  %MW1790   BLOCK28_END_TIME_H  "BLOCK28 End Time Hours - 14"
  %MW1791   BLOCK28_END_TIME_MN  "BLOCK28 End Time Minutes - 33"
  %MW1792   BLOCK28_SPARE_03
  %MW1793   BLOCK28_SPARE_04
  %MW1794   BLOCK28_RUNTIME_MN  "BLOCK28 Running Time for Cycle in Minutes"
  %MW1810   BLOCK29_START_TIME_Y  "BLOCK29 Start Time Years - 21"
  %MW1811   BLOCK29_START_TIME_M  "BLOCK29 Start Time  Months- 07"
  %MW1812   BLOCK29_START_TIME_D  "BLOCK29 Start Time Days- 19"
  %MW1813   BLOCK29_START_TIME_H  "BLOCK29 Start Time Hours - 14"
  %MW1814   BLOCK29_START_TIME_MN  "BLOCK29 Start Time Minutes - 33"
  %MW1815   BLOCK29_SPARE_01
  %MW1816   BLOCK29_SPARE_02
  %MW1817   BLOCK29_END_TIME_Y  "BLOCK29 End Time Years - 21"
  %MW1818   BLOCK29_END_TIME_M  "BLOCK29 End Time  Months- 07"
  %MW1819   BLOCK29_END_TIME_D  "BLOCK29 End Time Days- 19"
  %MW1820   BLOCK29_END_TIME_H  "BLOCK29 End Time Hours - 14"
  %MW1821   BLOCK29_END_TIME_MN  "BLOCK29 End Time Minutes - 33"
  %MW1822   BLOCK29_SPARE_03
  %MW1823   BLOCK29_SPARE_04
  %MW1824   BLOCK29_RUNTIME_MN  "BLOCK29 Running Time for Cycle in Minutes"
  %MW1840   BLOCK30_START_TIME_Y  "BLOCK30 Start Time Years - 21"
  %MW1841   BLOCK30_START_TIME_M  "BLOCK30 Start Time  Months- 07"
  %MW1842   BLOCK30_START_TIME_D  "BLOCK30 Start Time Days- 19"
  %MW1843   BLOCK30_START_TIME_H  "BLOCK30 Start Time Hours - 14"
  %MW1844   BLOCK30_START_TIME_MN  "BLOCK30 Start Time Minutes - 33"
  %MW1845   BLOCK30_SPARE_01
  %MW1846   BLOCK30_SPARE_02
  %MW1847   BLOCK30_END_TIME_Y  "BLOCK30 End Time Years - 21"
  %MW1848   BLOCK30_END_TIME_M  "BLOCK30 End Time  Months- 07"
  %MW1849   BLOCK30_END_TIME_D  "BLOCK30 End Time Days- 19"
  %MW1850   BLOCK30_END_TIME_H  "BLOCK30 End Time Hours - 14"
  %MW1851   BLOCK30_END_TIME_MN  "BLOCK30 End Time Minutes - 33"
  %MW1852   BLOCK30_SPARE_03
  %MW1853   BLOCK30_SPARE_04
  %MW1854   BLOCK30_RUNTIME_MN  "BLOCK30 Running Time for Cycle in Minutes"
  %MW2000   BLOCK2_1_ALARM  "Valve object alarm"
  %MW2001   BLOCK2_1_STATUS  "Valve object status"
  %MW2002   BLOCK2_1_TOTAL_FLOW  "Valve object total flow"
  %MW2500   ALARM_TEST
  %MW2501   STATUS_TEST
  %MW2502   TOTAL_FLOW_TEST
  %MW3000   EC_ALARM
  %MW3500   IRRI_ALARM
  %MW3501   IRRIGATION_STATUS
  %MW3502   IRRIGATION_TIME_LEFT
  %MW3503   BACKWASH_STATUS
  %MW3504   BACKWASH_TIME_LEFT
  %MW4000   TOTAL_WATER_FLOW
  %MF1012   BLOCK1_EC_SP  "BLOCK1 EC Setpoint"
  %MF1016   BLOCK1_TANK1_FLW_SP  "BLOCK1 Tank 1 Fertilizer Flow Setpoint"
  %MF1018   BLOCK1_TANK2_FLW_SP  "BLOCK1 Tank 2 Fertilizer Flow Setpoint"
  %MF1020   BLOCK1_TANK3_FLW_SP  "BLOCK1 Tank 3 Fertilizer Flow Setpoint"
  %MF1022   BLOCK1_TANK4_FLW_SP  "BLOCK1 Tank 4 Fertilizer Flow Setpoint"
  %MF1024   BLOCK1_TANK5_FLW_SP  "BLOCK1 Tank 5 Fertilizer Flow Setpoint"
  %MF1026   BLOCK1_TANK6_FLW_SP  "BLOCK1 Tank 6 Fertilizer Flow Setpoint"
  %MF1028   BLOCK1_TANK7_FLW_SP  "BLOCK1 Tank 7 Fertilizer Flow Setpoint"
  %MF1030   BLOCK1_TANK8_FLW_SP  "BLOCK1 Tank 8 Fertilizer Flow Setpoint"
  %MF1032   BLOCK1_TANK9_FLW_SP  "BLOCK1 Tank 9 Fertilizer Flow Setpoint"
  %MF1034   BLOCK1_TANK10_FLW_SP  "BLOCK1 Tank 10 Fertilizer Flow Setpoint"
  %MF1063   BLOCK2_EC_SP  "BLOCK2 EC Setpoint"
  %MF1067   BLOCK2_TANK1_FLW_SP  "BLOCK2 Tank 1 Fertilizer Flow Setpoint"
  %MF1069   BLOCK2_TANK2_FLW_SP  "BLOCK2 Tank 2 Fertilizer Flow Setpoint"
  %MF1071   BLOCK2_TANK3_FLW_SP  "BLOCK2 Tank 3 Fertilizer Flow Setpoint"
  %MF1073   BLOCK2_TANK4_FLW_SP  "BLOCK2 Tank 4 Fertilizer Flow Setpoint"
  %MF1075   BLOCK2_TANK5_FLW_SP  "BLOCK2 Tank 5 Fertilizer Flow Setpoint"
  %MF1077   BLOCK2_TANK6_FLW_SP  "BLOCK2 Tank 6 Fertilizer Flow Setpoint"
  %MF1079   BLOCK2_TANK7_FLW_SP  "BLOCK2 Tank 7 Fertilizer Flow Setpoint"
  %MF1081   BLOCK2_TANK8_FLW_SP  "BLOCK2 Tank 8 Fertilizer Flow Setpoint"
  %MF1083   BLOCK2_TANK9_FLW_SP  "BLOCK2 Tank 9 Fertilizer Flow Setpoint"
  %MF1085   BLOCK2_TANK10_FLW_SP  "BLOCK2 Tank 10 Fertilizer Flow Setpoint"
  %MF1114   BLOCK3_EC_SP  "BLOCK3 EC Setpoint"
  %MF1118   BLOCK3_TANK1_FLW_SP  "BLOCK3 Tank 1 Fertilizer Flow Setpoint"
  %MF1120   BLOCK3_TANK2_FLW_SP  "BLOCK3 Tank 2 Fertilizer Flow Setpoint"
  %MF1122   BLOCK3_TANK3_FLW_SP  "BLOCK3 Tank 3 Fertilizer Flow Setpoint"
  %MF1124   BLOCK3_TANK4_FLW_SP  "BLOCK3 Tank 4 Fertilizer Flow Setpoint"
  %MF1126   BLOCK3_TANK5_FLW_SP  "BLOCK3 Tank 5 Fertilizer Flow Setpoint"
  %MF1128   BLOCK3_TANK6_FLW_SP  "BLOCK3 Tank 6 Fertilizer Flow Setpoint"
  %MF1130   BLOCK3_TANK7_FLW_SP  "BLOCK3 Tank 7 Fertilizer Flow Setpoint"
  %MF1132   BLOCK3_TANK8_FLW_SP  "BLOCK3 Tank 8 Fertilizer Flow Setpoint"
  %MF1134   BLOCK3_TANK9_FLW_SP  "BLOCK3 Tank 9 Fertilizer Flow Setpoint"
  %MF1136   BLOCK3_TANK10_FLW_SP  "BLOCK3 Tank 10 Fertilizer Flow Setpoint"
  %MF1165   BLOCK4_EC_SP  "BLOCK4 EC Setpoint"
  %MF1169   BLOCK4_TANK1_FLW_SP  "BLOCK4 Tank 1 Fertilizer Flow Setpoint"
  %MF1171   BLOCK4_TANK2_FLW_SP  "BLOCK4 Tank 2 Fertilizer Flow Setpoint"
  %MF1173   BLOCK4_TANK3_FLW_SP  "BLOCK4 Tank 3 Fertilizer Flow Setpoint"
  %MF1175   BLOCK4_TANK4_FLW_SP  "BLOCK4 Tank 4 Fertilizer Flow Setpoint"
  %MF1177   BLOCK4_TANK5_FLW_SP  "BLOCK4 Tank 5 Fertilizer Flow Setpoint"
  %MF1179   BLOCK4_TANK6_FLW_SP  "BLOCK4 Tank 6 Fertilizer Flow Setpoint"
  %MF1181   BLOCK4_TANK7_FLW_SP  "BLOCK4 Tank 7 Fertilizer Flow Setpoint"
  %MF1183   BLOCK4_TANK8_FLW_SP  "BLOCK4 Tank 8 Fertilizer Flow Setpoint"
  %MF1185   BLOCK4_TANK9_FLW_SP  "BLOCK4 Tank 9 Fertilizer Flow Setpoint"
  %MF1187   BLOCK4_TANK10_FLW_SP  "BLOCK4 Tank 10 Fertilizer Flow Setpoint"
  %MF1216   BLOCK5_EC_SP  "BLOCK5 EC Setpoint"
  %MF1220   BLOCK5_TANK1_FLW_SP  "BLOCK5 Tank 1 Fertilizer Flow Setpoint"
  %MF1222   BLOCK5_TANK2_FLW_SP  "BLOCK5 Tank 2 Fertilizer Flow Setpoint"
  %MF1224   BLOCK5_TANK3_FLW_SP  "BLOCK5 Tank 3 Fertilizer Flow Setpoint"
  %MF1226   BLOCK5_TANK4_FLW_SP  "BLOCK5 Tank 4 Fertilizer Flow Setpoint"
  %MF1228   BLOCK5_TANK5_FLW_SP  "BLOCK5 Tank 5 Fertilizer Flow Setpoint"
  %MF1230   BLOCK5_TANK6_FLW_SP  "BLOCK5 Tank 6 Fertilizer Flow Setpoint"
  %MF1232   BLOCK5_TANK7_FLW_SP  "BLOCK5 Tank 7 Fertilizer Flow Setpoint"
  %MF1234   BLOCK5_TANK8_FLW_SP  "BLOCK5 Tank 8 Fertilizer Flow Setpoint"
  %MF1236   BLOCK5_TANK9_FLW_SP  "BLOCK5 Tank 9 Fertilizer Flow Setpoint"
  %MF1238   BLOCK5_TANK10_FLW_SP  "BLOCK5 Tank 10 Fertilizer Flow Setpoint"
  %MF1267   BLOCK6_EC_SP  "BLOCK6 EC Setpoint"
  %MF1271   BLOCK6_TANK1_FLW_SP  "BLOCK6 Tank 1 Fertilizer Flow Setpoint"
  %MF1273   BLOCK6_TANK2_FLW_SP  "BLOCK6 Tank 2 Fertilizer Flow Setpoint"
  %MF1275   BLOCK6_TANK3_FLW_SP  "BLOCK6 Tank 3 Fertilizer Flow Setpoint"
  %MF1277   BLOCK6_TANK4_FLW_SP  "BLOCK6 Tank 4 Fertilizer Flow Setpoint"
  %MF1279   BLOCK6_TANK5_FLW_SP  "BLOCK6 Tank 5 Fertilizer Flow Setpoint"
  %MF1281   BLOCK6_TANK6_FLW_SP  "BLOCK6 Tank 6 Fertilizer Flow Setpoint"
  %MF1283   BLOCK6_TANK7_FLW_SP  "BLOCK6 Tank 7 Fertilizer Flow Setpoint"
  %MF1285   BLOCK6_TANK8_FLW_SP  "BLOCK6 Tank 8 Fertilizer Flow Setpoint"
  %MF1287   BLOCK6_TANK9_FLW_SP  "BLOCK6 Tank 9 Fertilizer Flow Setpoint"
  %MF1289   BLOCK6_TANK10_FLW_SP  "BLOCK6 Tank 10 Fertilizer Flow Setpoint"
  %MF1318   BLOCK7_EC_SP  "BLOCK7 EC Setpoint"
  %MF1322   BLOCK7_TANK1_FLW_SP  "BLOCK7 Tank 1 Fertilizer Flow Setpoint"
  %MF1324   BLOCK7_TANK2_FLW_SP  "BLOCK7 Tank 2 Fertilizer Flow Setpoint"
  %MF1326   BLOCK7_TANK3_FLW_SP  "BLOCK7 Tank 3 Fertilizer Flow Setpoint"
  %MF1328   BLOCK7_TANK4_FLW_SP  "BLOCK7 Tank 4 Fertilizer Flow Setpoint"
  %MF1330   BLOCK7_TANK5_FLW_SP  "BLOCK7 Tank 5 Fertilizer Flow Setpoint"
  %MF1332   BLOCK7_TANK6_FLW_SP  "BLOCK7 Tank 6 Fertilizer Flow Setpoint"
  %MF1334   BLOCK7_TANK7_FLW_SP  "BLOCK7 Tank 7 Fertilizer Flow Setpoint"
  %MF1336   BLOCK7_TANK8_FLW_SP  "BLOCK7 Tank 8 Fertilizer Flow Setpoint"
  %MF1338   BLOCK7_TANK9_FLW_SP  "BLOCK7 Tank 9 Fertilizer Flow Setpoint"
  %MF1340   BLOCK7_TANK10_FLW_SP  "BLOCK7 Tank 10 Fertilizer Flow Setpoint"
  %MF1369   BLOCK8_EC_SP  "BLOCK8 EC Setpoint"
  %MF1373   BLOCK8_TANK1_FLW_SP  "BLOCK8 Tank 1 Fertilizer Flow Setpoint"
  %MF1375   BLOCK8_TANK2_FLW_SP  "BLOCK8 Tank 2 Fertilizer Flow Setpoint"
  %MF1377   BLOCK8_TANK3_FLW_SP  "BLOCK8 Tank 3 Fertilizer Flow Setpoint"
  %MF1379   BLOCK8_TANK4_FLW_SP  "BLOCK8 Tank 4 Fertilizer Flow Setpoint"
  %MF1381   BLOCK8_TANK5_FLW_SP  "BLOCK8 Tank 5 Fertilizer Flow Setpoint"
  %MF1383   BLOCK8_TANK6_FLW_SP  "BLOCK8 Tank 6 Fertilizer Flow Setpoint"
  %MF1385   BLOCK8_TANK7_FLW_SP  "BLOCK8 Tank 7 Fertilizer Flow Setpoint"
  %MF1387   BLOCK8_TANK8_FLW_SP  "BLOCK8 Tank 8 Fertilizer Flow Setpoint"
  %MF1389   BLOCK8_TANK9_FLW_SP  "BLOCK8 Tank 9 Fertilizer Flow Setpoint"
  %MF1391   BLOCK8_TANK10_FLW_SP  "BLOCK8 Tank 10 Fertilizer Flow Setpoint"
  %MF1420   BLOCK9_EC_SP  "BLOCK9 EC Setpoint"
  %MF1424   BLOCK9_TANK1_FLW_SP  "BLOCK9 Tank 1 Fertilizer Flow Setpoint"
  %MF1426   BLOCK9_TANK2_FLW_SP  "BLOCK9 Tank 2 Fertilizer Flow Setpoint"
  %MF1428   BLOCK9_TANK3_FLW_SP  "BLOCK9 Tank 3 Fertilizer Flow Setpoint"
  %MF1430   BLOCK9_TANK4_FLW_SP  "BLOCK9 Tank 4 Fertilizer Flow Setpoint"
  %MF1432   BLOCK9_TANK5_FLW_SP  "BLOCK9 Tank 5 Fertilizer Flow Setpoint"
  %MF1434   BLOCK9_TANK6_FLW_SP  "BLOCK9 Tank 6 Fertilizer Flow Setpoint"
  %MF1436   BLOCK9_TANK7_FLW_SP  "BLOCK9 Tank 7 Fertilizer Flow Setpoint"
  %MF1438   BLOCK9_TANK8_FLW_SP  "BLOCK9 Tank 8 Fertilizer Flow Setpoint"
  %MF1440   BLOCK9_TANK9_FLW_SP  "BLOCK9 Tank 9 Fertilizer Flow Setpoint"
  %MF1442   BLOCK9_TANK10_FLW_SP  "BLOCK9 Tank 10 Fertilizer Flow Setpoint"
  %MF1471   BLOCK10_EC_SP  "BLOCK10 EC Setpoint"
  %MF1475   BLOCK10_TANK1_FLW_SP  "BLOCK10 Tank 1 Fertilizer Flow Setpoint"
  %MF1477   BLOCK10_TANK2_FLW_SP  "BLOCK10 Tank 2 Fertilizer Flow Setpoint"
  %MF1479   BLOCK10_TANK3_FLW_SP  "BLOCK10 Tank 3 Fertilizer Flow Setpoint"
  %MF1481   BLOCK10_TANK4_FLW_SP  "BLOCK10 Tank 4 Fertilizer Flow Setpoint"
  %MF1483   BLOCK10_TANK5_FLW_SP  "BLOCK10 Tank 5 Fertilizer Flow Setpoint"
  %MF1485   BLOCK10_TANK6_FLW_SP  "BLOCK10 Tank 6 Fertilizer Flow Setpoint"
  %MF1487   BLOCK10_TANK7_FLW_SP  "BLOCK10 Tank 7 Fertilizer Flow Setpoint"
  %MF1489   BLOCK10_TANK8_FLW_SP  "BLOCK10 Tank 8 Fertilizer Flow Setpoint"
  %MF1491   BLOCK10_TANK9_FLW_SP  "BLOCK10 Tank 9 Fertilizer Flow Setpoint"
  %MF1493   BLOCK10_TANK10_FLW_SP  "BLOCK10 Tank 10 Fertilizer Flow Setpoint"
  %MF1522   BLOCK11_EC_SP  "BLOCK11 EC Setpoint"
  %MF1526   BLOCK11_TANK1_FLW_SP  "BLOCK11 Tank 1 Fertilizer Flow Setpoint"
  %MF1528   BLOCK11_TANK2_FLW_SP  "BLOCK11 Tank 2 Fertilizer Flow Setpoint"
  %MF1530   BLOCK11_TANK3_FLW_SP  "BLOCK11 Tank 3 Fertilizer Flow Setpoint"
  %MF1532   BLOCK11_TANK4_FLW_SP  "BLOCK11 Tank 4 Fertilizer Flow Setpoint"
  %MF1534   BLOCK11_TANK5_FLW_SP  "BLOCK11 Tank 5 Fertilizer Flow Setpoint"
  %MF1536   BLOCK11_TANK6_FLW_SP  "BLOCK11 Tank 6 Fertilizer Flow Setpoint"
  %MF1538   BLOCK11_TANK7_FLW_SP  "BLOCK11 Tank 7 Fertilizer Flow Setpoint"
  %MF1540   BLOCK11_TANK8_FLW_SP  "BLOCK11 Tank 8 Fertilizer Flow Setpoint"
  %MF1542   BLOCK11_TANK9_FLW_SP  "BLOCK11 Tank 9 Fertilizer Flow Setpoint"
  %MF1544   BLOCK11_TANK10_FLW_SP  "BLOCK11 Tank 10 Fertilizer Flow Setpoint"
  %MF1573   BLOCK12_EC_SP  "BLOCK12 EC Setpoint"
  %MF1577   BLOCK12_TANK1_FLW_SP  "BLOCK12 Tank 1 Fertilizer Flow Setpoint"
  %MF1579   BLOCK12_TANK2_FLW_SP  "BLOCK12 Tank 2 Fertilizer Flow Setpoint"
  %MF1581   BLOCK12_TANK3_FLW_SP  "BLOCK12 Tank 3 Fertilizer Flow Setpoint"
  %MF1583   BLOCK12_TANK4_FLW_SP  "BLOCK12 Tank 4 Fertilizer Flow Setpoint"
  %MF1585   BLOCK12_TANK5_FLW_SP  "BLOCK12 Tank 5 Fertilizer Flow Setpoint"
  %MF1587   BLOCK12_TANK6_FLW_SP  "BLOCK12 Tank 6 Fertilizer Flow Setpoint"
  %MF1589   BLOCK12_TANK7_FLW_SP  "BLOCK12 Tank 7 Fertilizer Flow Setpoint"
  %MF1591   BLOCK12_TANK8_FLW_SP  "BLOCK12 Tank 8 Fertilizer Flow Setpoint"
  %MF1593   BLOCK12_TANK9_FLW_SP  "BLOCK12 Tank 9 Fertilizer Flow Setpoint"
  %MF1595   BLOCK12_TANK10_FLW_SP  "BLOCK12 Tank 10 Fertilizer Flow Setpoint"
  %MF1624   BLOCK13_EC_SP  "BLOCK13 EC Setpoint"
  %MF1628   BLOCK13_TANK1_FLW_SP  "BLOCK13 Tank 1 Fertilizer Flow Setpoint"
  %MF1630   BLOCK13_TANK2_FLW_SP  "BLOCK13 Tank 2 Fertilizer Flow Setpoint"
  %MF1632   BLOCK13_TANK3_FLW_SP  "BLOCK13 Tank 3 Fertilizer Flow Setpoint"
  %MF1634   BLOCK13_TANK4_FLW_SP  "BLOCK13 Tank 4 Fertilizer Flow Setpoint"
  %MF1636   BLOCK13_TANK5_FLW_SP  "BLOCK13 Tank 5 Fertilizer Flow Setpoint"
  %MF1638   BLOCK13_TANK6_FLW_SP  "BLOCK13 Tank 6 Fertilizer Flow Setpoint"
  %MF1640   BLOCK13_TANK7_FLW_SP  "BLOCK13 Tank 7 Fertilizer Flow Setpoint"
  %MF1642   BLOCK13_TANK8_FLW_SP  "BLOCK13 Tank 8 Fertilizer Flow Setpoint"
  %MF1644   BLOCK13_TANK9_FLW_SP  "BLOCK13 Tank 9 Fertilizer Flow Setpoint"
  %MF1646   BLOCK13_TANK10_FLW_SP  "BLOCK13 Tank 10 Fertilizer Flow Setpoint"
  %MF1675   BLOCK14_EC_SP  "BLOCK14 EC Setpoint"
  %MF1679   BLOCK14_TANK1_FLW_SP  "BLOCK14 Tank 1 Fertilizer Flow Setpoint"
  %MF1681   BLOCK14_TANK2_FLW_SP  "BLOCK14 Tank 2 Fertilizer Flow Setpoint"
  %MF1683   BLOCK14_TANK3_FLW_SP  "BLOCK14 Tank 3 Fertilizer Flow Setpoint"
  %MF1685   BLOCK14_TANK4_FLW_SP  "BLOCK14 Tank 4 Fertilizer Flow Setpoint"
  %MF1687   BLOCK14_TANK5_FLW_SP  "BLOCK14 Tank 5 Fertilizer Flow Setpoint"
  %MF1689   BLOCK14_TANK6_FLW_SP  "BLOCK14 Tank 6 Fertilizer Flow Setpoint"
  %MF1691   BLOCK14_TANK7_FLW_SP  "BLOCK14 Tank 7 Fertilizer Flow Setpoint"
  %MF1693   BLOCK14_TANK8_FLW_SP  "BLOCK14 Tank 8 Fertilizer Flow Setpoint"
  %MF1695   BLOCK14_TANK9_FLW_SP  "BLOCK14 Tank 9 Fertilizer Flow Setpoint"
  %MF1697   BLOCK14_TANK10_FLW_SP  "BLOCK14 Tank 10 Fertilizer Flow Setpoint"
  %MF1726   BLOCK15_EC_SP  "BLOCK15 EC Setpoint"
  %MF1730   BLOCK15_TANK1_FLW_SP  "BLOCK15 Tank 1 Fertilizer Flow Setpoint"
  %MF1732   BLOCK15_TANK2_FLW_SP  "BLOCK15 Tank 2 Fertilizer Flow Setpoint"
  %MF1734   BLOCK15_TANK3_FLW_SP  "BLOCK15 Tank 3 Fertilizer Flow Setpoint"
  %MF1736   BLOCK15_TANK4_FLW_SP  "BLOCK15 Tank 4 Fertilizer Flow Setpoint"
  %MF1738   BLOCK15_TANK5_FLW_SP  "BLOCK15 Tank 5 Fertilizer Flow Setpoint"
  %MF1740   BLOCK15_TANK6_FLW_SP  "BLOCK15 Tank 6 Fertilizer Flow Setpoint"
  %MF1742   BLOCK15_TANK7_FLW_SP  "BLOCK15 Tank 7 Fertilizer Flow Setpoint"
  %MF1744   BLOCK15_TANK8_FLW_SP  "BLOCK15 Tank 8 Fertilizer Flow Setpoint"
  %MF1746   BLOCK15_TANK9_FLW_SP  "BLOCK15 Tank 9 Fertilizer Flow Setpoint"
  %MF1748   BLOCK15_TANK10_FLW_SP  "BLOCK15 Tank 10 Fertilizer Flow Setpoint"
  %MF2004   BLOCK2_1_RT_FLOW  "Alarm object real time flow"
  %MF2504   REAL_TIME_FLOW_TEST
  %MF2506   REAL_TIME_PRESSURE_TEST
  %MF3002   EC_VALUE
  %MF3004   EC_AVG_VALUE
  %MF3006   EC_SETPOINT
  %MF3506   IRRIGATION_PERCENTAGE_LEFT
  %MF3508   BACKWASH_PERCENTAGE_LEFT
  %MF4010   TOTAL_FERTILIZER_01
  %MF4018   TOTAL_FERTILIZER_05
  %MF4030   TOTAL_PLACEHOLDER_01
  %MF4034   TOTAL_PLACEHOLDER_03

POU New POU
  (* SectionNumber=1 *)

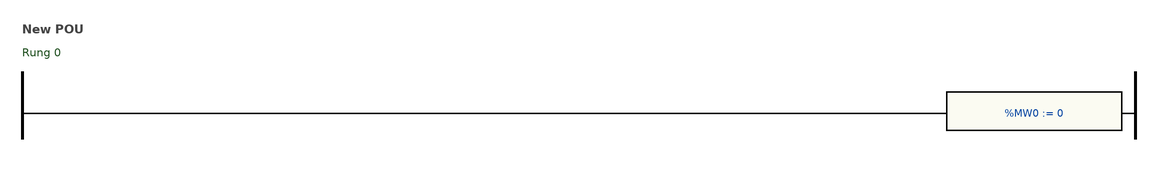

// Rung 0
  LD 1
  [ %MW0 := 0 ]
  // as ST:
  //   %MW0 := 0;
